// TIA Portal V21 export
DATA_BLOCK "Matrice"   // DB35
{ S7_Optimized_Access := 'TRUE' }
// stored: MemoryReserve 100
   VAR
      K_Linea : Array[0..30] of Int;
      K_Colonna : Array[0..50] of Int;
      Hmi : Struct
         IndicePrimoKLinea : Int := 1;
         IndicePrimoKColonna : Int := 1;
         AbilitaScrollAvanti_Linea : Bool := TRUE;
         AbilitaScrollIndietro_Linea : Bool := FALSE;
         AbilitaScrollAvanti_Colonna : Bool := TRUE;
         AbilitaScrollIndietro_Colonna : Bool := FALSE;
         AggiornaMatrice : Bool := FALSE;
         NuovoPercorso : Struct
            SelezioneNuovoPercorso : Bool := FALSE;
            DeselezioneNuovoPercorso : Bool := FALSE;
            Sorgente : Int := 0;
            Destinazione : Int := 0;
            AbilitaSceltaSorgente : Bool := FALSE;
            AbilitaSceltaDestinazione : Array[0.."K_NumStazione"] of Bool;
         END_STRUCT;
      END_STRUCT;
      PercorsoSelezionato : Array[0..27, 0..50] of Int;
   END_VAR
BEGIN
   K_Linea[0..30] := 0;
   K_Colonna[0..50] := 0;
   Hmi.NuovoPercorso.AbilitaSceltaDestinazione[0..1] := FALSE;
   PercorsoSelezionato[0,0..49] := 2;
   PercorsoSelezionato[0,50] := 0;
   PercorsoSelezionato[1,0..50] := 0;
   PercorsoSelezionato[2,0..50] := 0;
   PercorsoSelezionato[3,0..50] := 0;
   PercorsoSelezionato[4,0..50] := 0;
   PercorsoSelezionato[5,0..50] := 0;
   PercorsoSelezionato[6,0..50] := 0;
   PercorsoSelezionato[7,0..50] := 0;
   PercorsoSelezionato[8,0..50] := 0;
   PercorsoSelezionato[9,0..50] := 0;
   PercorsoSelezionato[10,0..50] := 0;
   PercorsoSelezionato[11,0..50] := 0;
   PercorsoSelezionato[12,0..50] := 0;
   PercorsoSelezionato[13,0..50] := 0;
   PercorsoSelezionato[14,0..50] := 0;
   PercorsoSelezionato[15,0..50] := 0;
   PercorsoSelezionato[16,0..50] := 0;
   PercorsoSelezionato[17,0..50] := 0;
   PercorsoSelezionato[18,0..50] := 0;
   PercorsoSelezionato[19,0..50] := 0;
   PercorsoSelezionato[20,0..50] := 0;
   PercorsoSelezionato[21,0..50] := 0;
   PercorsoSelezionato[22,0..50] := 0;
   PercorsoSelezionato[23,0..50] := 0;
   PercorsoSelezionato[24,0..50] := 0;
   PercorsoSelezionato[25,0..50] := 0;
   PercorsoSelezionato[26,0..50] := 0;
   PercorsoSelezionato[27,0..50] := 0;
END_DATA_BLOCK
